FUNCTION_BLOCK FB_CassetteLoader EXTENDS FB_PackML_BaseModule

VAR
	    // Sub module definitions here

    // List of sub modules
    ipSubModules_Init : ARRAY[1..Parameters_PackML_Base.MAX_NO_OF_SUBMODULES] OF I_PackML_BaseModule := [];

    // Component definitions here
    ElevatorAxisA : FB_Component_BasicAxis := (Name := 'ElevatorA');
	ElevatorAxisB : FB_Component_BasicAxis := (Name := 'ElevatorB');
	ShuttleAxis : FB_Component_BasicAxis := (Name := 'Shuttle');
	MapSensorA : FB_DigitalSensor := (Name := 'MapSensorA');
	MapSensorB : FB_DigitalSensor := (Name := 'MapSensorB');
	
	//Assign Homing Routine to Use the Absolute Encoder, using the persistent struct below
	AbsHomingElevA : FB_HomeRoutine_AbsHoming;
	AbsHomingElevB : FB_HomeRoutine_AbsHoming;
	AbsHomingShuttle : FB_HomeRoutine_AbsHoming;
		
	//Alarms for this Module
	LoaderAlarms : ARRAY[1..LOADER_ALARM_COUNT] OF FB_TcAlarm;
	
	//Data for module
    Recipe : ST_LoaderRecipe;
	CassetteAStatus : ST_CassetteStatus;
	CassetteBStatus : ST_CassetteStatus;
	_ElevatorAxisAStagePosition : LREAL;
	_ElevatorAxisBStagePosition : LREAL;
	_ShuttleAxisStagePosition : LREAL;
	_ElevatorAxisAHomePosition : LREAL;
	_ElevatorAxisBHomePosition : LREAL;
	_ShuttleAxisHomePosition : LREAL;
	
	//HMI Control for EM
    fbControlSourceHMI : FB_ControlSource_HMI;
	
	//Load or Unload Mode: Commanded by External, TRUE= Load, FALSE = Unload
	_LoadOrUnload : BOOL;
	_ShuttleReady : BOOL;

	//This trigger each axis at the abs zero position when in maintenance or manual mode
	AbsHomeCmdA: BOOL;
	AbsHomeCmdB: BOOL;
	AbsHomeCmdShuttle: BOOL;
	_NeedsMapping: BOOL;
	_NextSlot: DINT;
	_NextCassette: INT;
END_VAR

VAR CONSTANT
	LOADER_ALARM_COUNT : INT := 6;
END_VAR

VAR PERSISTENT
	ElevAHomingParameters : ST_AbsHomeParameters;
	ElevBHomingParameters : ST_AbsHomeParameters;
	ShuttleHomingParameters : ST_AbsHomeParameters;
END_VAR

ShuttleHomingParameters.PositionBias := 0;

METHOD PROTECTED Aborting
VAR_INPUT
END_VAR
CASE SequenceState OF
    0:
        NoStateTasksToComplete := FALSE;
        SequenceState          := SequenceState + 10;
    10:
        ElevatorAxisA.Stop();
		ElevatorAxisB.Stop();
		ShuttleAxis.Stop();
//        IF (ElevatorAxisA.Stopped AND ElevatorAxisB.Stopped AND ShuttleAxis.Stopped) THEN
//            SequenceState := SequenceState + 10;
//        END_IF
		SequenceState := SequenceState + 10;
    20:
        // Disable here
        ElevatorAxisA.Disable();
		ElevatorAxisB.Disable();
		ShuttleAxis.Disable();

        // Check not enabled here
        IF NOT (ElevatorAxisA.Enabled AND ElevatorAxisB.Enabled AND ShuttleAxis.Enabled) THEN
            SequenceState := SequenceState + 10;
        END_IF
    30:
        StateTasksComplete := TRUE;
END_CASE

SUPER^.Aborting();
END_METHOD

PROPERTY BladeThickness : LREAL
GET
BladeThickness := recipe.Elevator.BladeThickness;
END_GET
SET
BladeThickness := recipe.Elevator.BladeThickness;
END_SET
END_PROPERTY

PROPERTY CassettePitch : LREAL
GET
CassettePitch := recipe.Elevator.CassettePitch;
END_GET
SET
recipe.Elevator.CassettePitch := CassettePitch;
END_SET
END_PROPERTY

PROPERTY CassetteSlotHeight : LREAL
GET
CassetteSlotHeight := recipe.Elevator.CassetteSlotHeight;
END_GET
SET
recipe.Elevator.CassetteSlotHeight := CassetteSlotHeight;
END_SET
END_PROPERTY

PROPERTY CassetteSlotNumber : INT
GET
CassetteSlotNumber := recipe.Elevator.CassetteSlotNumber;
END_GET
SET
recipe.Elevator.CassetteSlotNumber := CassetteSlotNumber;
END_SET
END_PROPERTY

METHOD PROTECTED Clearing
VAR_INPUT
END_VAR
CASE SequenceState OF
    0:
        NoStateTasksToComplete := FALSE;
        SequenceState          := SequenceState + 10;
	10:
        //Reset any alarms that get latched
        //PullWheelAlarms[E_PullWheels.StartTimeout].Clear(0, 0);
        SequenceState := SequenceState + 10;
    20:
        StateTasksComplete := TRUE;
END_CASE

SUPER^.Clearing();
END_METHOD

METHOD CyclicLogic
VAR_INPUT
END_VAR

VAR
	i : INT;
	TotalInCassetteA : INT;
	TotalInCassetteB : INT;
	CassetteAInteger : ARRAY[0..23] OF INT; //matching array with INT type
	CassetteBInteger : ARRAY[0..23] OF INT; //matching array with INT type
END_VAR
IF NOT _InitComplete THEN
    _InitComplete := Initialize();
    RETURN;
END_IF

SUPER^.CyclicLogic();

//Set the current alarm severity for this module
_CurrentAlarmSeverity   := F_GetMaxSeverityRaised(Alarms := LoaderAlarms, CurrentSeverity := _CurrentAlarmSeverity);

//Add up the number of waveguides in each cassette and mark the cassette status as full
	FOR i := 0 TO 23 DO
		IF CassetteAStatus.WaveguidePresent[i] = TRUE THEN
			CassetteAInteger[i] := 1;
		ELSE
			CassetteAInteger[i] := 0;
		END_IF
		TotalInCassetteA := TotalInCassetteA + CassetteAInteger[i];
		IF TotalInCassetteA > 22 THEN
			CassetteAStatus.CassetteFull := TRUE;
		END_IF
	END_FOR; 
	
	FOR i := 0 TO 23 DO
		IF CassetteBStatus.WaveguidePresent[i] = TRUE THEN
			CassetteBInteger[i] := 1;
		ELSE
			CassetteBInteger[i] := 0;
		END_IF
		TotalInCassetteB := TotalInCassetteB + CassetteBInteger[i];
		IF TotalInCassetteB > 22 THEN
			CassetteBStatus.CassetteFull := TRUE;
		END_IF
	END_FOR;
END_METHOD

METHOD DetermineNextSlot : DINT
VAR_INPUT
	CassetteID : ST_CassetteStatus;
END_VAR

VAR
	i: DINT;
END_VAR
//This method searches the wafer map array from the bottom to the top, returning the highest slot that is empty
	FOR i := 0 TO 23 DO
		IF CassetteID.WaveguidePresent[i] = FALSE THEN
			DetermineNextSlot := i;
		END_IF
	END_FOR;
END_METHOD

METHOD DetermineNextWaveguide : INT
VAR_INPUT
		CassetteID : ST_CassetteStatus;
END_VAR

VAR
	i: INT;
END_VAR
//This method searches the wafer map array from the bottom to the top, returning the lowest slot that is full
	FOR i := 23 TO 0 DO
		IF CassetteID.WaveguidePresent[i] = TRUE THEN
			DetermineNextWaveguide := i;
		END_IF
	END_FOR;
END_METHOD

PROPERTY ElevatorAcceleration : LREAL
GET
ElevatorAcceleration := recipe.Elevator.Acceleration;
END_GET
SET
recipe.Elevator.Acceleration := ElevatorAcceleration;
END_SET
END_PROPERTY

PROPERTY ElevatorFirstWaveguidePosition : LREAL
GET
ElevatorFirstWaveguidePosition := recipe.Elevator.FirstWaveguidePosition;
END_GET
SET
recipe.Elevator.FirstWaveguidePosition := ElevatorFirstWaveguidePosition;
END_SET
END_PROPERTY

PROPERTY ElevatorVelocity : LREAL
GET
ElevatorVelocity := recipe.Elevator.Velocity;
END_GET
SET
recipe.Elevator.Velocity := ElevatorVelocity;
END_SET
END_PROPERTY

METHOD PROTECTED Execute
VAR_INPUT
END_VAR
CASE _CurrentMode OF
    //=================================PRODUCTION MODE==================================
    E_PMLUnitMode.ePMLUnitMode_Production:
		IF _LoadOrUnload = TRUE THEN // _LoadOrUnload = TRUE means LOAD the cassette
			
		//Loading case
			CASE SequenceState OF

				10:		//Figure out where to put the next waveguide
						//we will load cassette A (top-down) before cassette B (top-down), so if A is full start loading B 
						IF NOT CassetteAStatus.CassetteFull THEN
							_NextSlot := DetermineNextSlot(CassetteID := CassetteAStatus);
							_NextCassette := 0; 
						ELSE	
							_NextSlot := DetermineNextSlot(CassetteID := CassetteBStatus);
							_NextCassette := 1;
						END_IF
						SequenceState := SequenceState + 10;
				20:		//Make sure that the space under/over the slot is clear, abort if obstructed
						IF _NextCassette = 0 THEN
							IF (CassetteAStatus.ClearBelowWaveguide[_NextSlot] AND CassetteAStatus.ClearBelowWaveguide[_NextSlot + 1]) = TRUE THEN
								SequenceState := SequenceState + 10;
							ELSE
								//changestate(ePMLState_Aborting);
							END_IF
						ELSE
							IF (CassetteBStatus.ClearBelowWaveguide[_NextSlot] AND CassetteBStatus.ClearBelowWaveguide[_NextSlot + 1]) = TRUE THEN
								SequenceState := SequenceState + 10;
							ELSE
								//changestate(ePMLState_Aborting);
							END_IF
						END_IF
						SequenceState := SequenceState + 10;
				30: 	//Move all to staged position
						SequenceState := SequenceState + 10;
				40:		//Call PlaceToNextOpenSlot method
						PlaceToNextOpenSlot(_NextCassette, _NextSlot);
						SequenceState := SequenceState + 10;
				50:		//Depending on which cassette we loaded, update the map to add the waveguide:
						IF _NextCassette = 0 THEN
							CassetteAStatus.WaveguidePresent[_NextSlot]:= 1;
						ELSE
							CassetteBStatus.WaveguidePresent[_NextSlot]:= 1;
						END_IF
						SequenceState := SequenceState + 10;

				99:		//based on the cassette status, either go into suspending or completing
						IF (CassetteAStatus.CassetteFull AND CassetteBStatus.CassetteFull) THEN
							StateComplete();
						ELSE
							//go into suspending state
							//changestate(ePMLState_Suspending);
						END_IF
			END_CASE
			
		//Unload Case	
		ELSE //_LoadOrUnload = FALSE means UNLOAD the cassette
			
			CASE SequenceState OF
				10: //Figure out which waveguide to remove first
				//we will unload cassette A (bottom-up) before cassette B (bottom-up), so if A is empty start unloading B
						IF CassetteAStatus.CassetteFull THEN
							_NextSlot := DetermineNextWaveguide(CassetteID := CassetteAStatus);
							_NextCassette := 0; 
						ELSE	
							_NextSlot := DetermineNextWaveguide(CassetteID := CassetteBStatus);
							_NextCassette := 1;
						END_IF
						SequenceState := SequenceState + 10;
				20:		//Make sure that the space under/over the slot is clear, abort if obstructed
						IF _NextCassette = 0 THEN
							IF (CassetteAStatus.ClearBelowWaveguide[_NextSlot] AND CassetteAStatus.ClearBelowWaveguide[_NextSlot + 1]) = TRUE THEN
								SequenceState := SequenceState + 10;
							ELSE
								//changestate(ePMLState_Aborting);
							END_IF
						ELSE
							IF (CassetteBStatus.ClearBelowWaveguide[_NextSlot] AND CassetteBStatus.ClearBelowWaveguide[_NextSlot + 1]) = TRUE THEN
								SequenceState := SequenceState + 10;
							ELSE
								//changestate(ePMLState_Aborting);
							END_IF
						END_IF
						SequenceState := SequenceState + 10;
				30:		//Pre-position the stages
						IF _NextCassette = 0 THEN
							ElevatorAxisA.MoveAbsolute(_ElevatorAxisAStagePosition,TRUE);
							ElevatorAxisB.MoveAbsolute(_ElevatorAxisBHomePosition,TRUE);
							ShuttleAxis.MoveAbsolute(_ShuttleAxisStagePosition, TRUE);
						ELSE
							ElevatorAxisA.MoveAbsolute(_ElevatorAxisAHomePosition,TRUE);
							ElevatorAxisB.MoveAbsolute(_ElevatorAxisBStagePosition,TRUE);
							ShuttleAxis.MoveAbsolute(_ShuttleAxisStagePosition, TRUE);
						END_IF
						SequenceState := SequenceState + 10;
				40: 	//Confirm all axis preposition movements are complete
						IF (ElevatorAxisA.Busy AND ElevatorAxisB.Busy AND ShuttleAxis.Busy) THEN
							SequenceState := SequenceState + 10;
						END_IF
				50:		//Call GetNextWaveguide method
						GetNextWaveGuide(_NextCassette, _NextSlot);
						SequenceState := SequenceState + 10;
				60:		//Depending on which cassette we unloaded, update the map to remove the waveguide:
						IF _NextCassette = 0 THEN
							CassetteAStatus.WaveguidePresent[_NextSlot]:= 0;
						ELSE
							CassetteBStatus.WaveguidePresent[_NextSlot]:= 0;
						END_IF
						SequenceState := SequenceState + 10;
				
			END_CASE
		END_IF
//If we are waiting for the tool to load/unload the waveguide, switch to Suspending state



    //=================================MAINTENANCE & MANUAL MODE==================================		
    E_PMLUnitMode.ePMLUnitMode_Maintenance, E_PMLUnitMode.ePMLUnitMode_Manual:
        //Reset the abs zero position when commanded
		IF AbsHomeCmdA THEN
    		AbsHomingElevA.Execute();
    		AbsHomeCmdA:=FALSE;
		END_IF;
		
		IF AbsHomeCmdB THEN
    		AbsHomingElevA.Execute();
    		AbsHomeCmdB:=FALSE;
		END_IF;
		
		IF AbsHomeCmdShuttle THEN
    		AbsHomingElevA.Execute();
    		AbsHomeCmdShuttle:=FALSE;
		END_IF;
END_CASE
END_METHOD

METHOD GetNextWaveguide : BOOL
VAR_INPUT
	NextCassette : INT;
	NextSlot : DINT;
END_VAR
//This method will get the waveguide in the cassette and slot defined as next-available and move the shuttle to the tool position
END_METHOD

//! @summary Basic module initialization logic
METHOD PROTECTED Initialize : BOOL;
VAR
	i						 : UDINT;
	varInfo					 : __SYSTEM.VAR_INFO;
	AllSubUnitsInitialized	 : BOOL := TRUE;
	AllComponentsInitialized : BOOL := TRUE;
END_VAR

//! @description This method is called by <c>CyclicLogic()</c> as required
Initialize := FALSE;
CASE DescendantSequenceState OF
    0:
		//RegisterComponent here (none for now)
        _LogModeChanges         := FALSE;
        _LogStateChanges        := FALSE;
        DescendantSequenceState := DescendantSequenceState + 10;
    10:
        //Setup Custom modes here
        CustomModes(eMode                          :=,
                    sName                          := 'Name',
                    bDisableClearing               := FALSE,
                    bDisableStarting               := FALSE,
                    bDisableSuspended              := FALSE,
                    bDisableStopping               := FALSE,
                    bDisableAborting               := FALSE,
                    bDisableHolding                := TRUE, //no operator hold state 
                    bDisableHeld                   := TRUE,
                    bDisableUnholding              := TRUE,
                    bDisableSuspending             := FALSE,
                    bDisableUnsuspending           := FALSE,
                    bDisableResetting              := FALSE,
                    bDisableIdle                   := FALSE,
                    bDisableCompleting             := FALSE,
                    bDisableComplete               := FALSE,
                    bEnableUnitModeChangeStopped   := TRUE,
                    bEnableUnitModeChangeIdle      := TRUE,
                    bEnableUnitModeChangeSuspended := FALSE,
                    bEnableUnitModeChangeExecute   := FALSE,
                    bEnableUnitModeChangeAborted   := FALSE,
                    bEnableUnitModeChangeHeld      := FALSE,
                    bEnableUnitModeChangeComplete  := FALSE,
                    bError                         =>,
                    nErrorId                       =>);
        DescendantSequenceState := DescendantSequenceState + 10;
    20:
        //Copy Mode names
        FOR i := 1 TO 3 DO
            ModeNames[i] := F_UnitModeToString(UDINT_TO_DINT(i));
        END_FOR

        //Initialize_TagData();
		RegisterExternalController(Controller := fbControlSourceHMI);
		fbControlSourceHMI.CyclicLogic();
        DescendantSequenceState := DescendantSequenceState + 10;
		
	30: //Register homing methods for each axis
//				ShuttleAxis.HomeMethod := AbsHomingShuttle;
//				AbsHomingShuttle.Parameters := ShuttleHomingParameters;
//				ElevatorAxisA.HomeMethod := AbsHomingElevA;
//				AbsHomingElevA.Parameters := ElevAHomingParameters;
//				ElevatorAxisB.HomeMethod := AbsHomingElevB;
//				AbsHomingElevB.Parameters := ElevBHomingParameters;
      	DescendantSequenceState := DescendantSequenceState + 10;
    40:
        //Call the Super
        IF SUPER^.Initialize() THEN
            DescendantSequenceState := DescendantSequenceState + 10;
        END_IF
    50:
        Initialize := TRUE;
END_CASE
END_METHOD

METHOD LoadCassette : BOOL
VAR_INPUT

END_VAR
(* This method will allow the user to stop the machine, open the door, install cassettes, 
close the door, restart the machine, map the cassettes and go into a ready state *)
END_METHOD

PROPERTY LoadOrUnload : bool
GET
LoadOrUnload := _LoadOrUnload;
END_GET
SET
_LoadOrUnload := LoadOrUnload;
END_SET
END_PROPERTY

METHOD MapCassette : BOOL
VAR_INPUT
	CassetteToMap : INT; //Cassette A is zero, Cassette B is one, etc.
END_VAR

VAR
	
END_VAR

//this method will map the cassette specified in CassetteToMap, saving the output in the array CassetteAStatus.WaveguidePresent
END_METHOD

METHOD PlaceToNextOpenSlot : BOOL
VAR_INPUT
	NextCassette : INT;
	NextSlot : DINT;
END_VAR
//This method will place the waveguide (placed on the blade by the tool) to the next open slot
END_METHOD

METHOD PROTECTED Resetting
VAR_INPUT
END_VAR
CASE _CurrentMode OF
    //=================================PRODUCTION MODE==================================
    E_PMLUnitMode.ePMLUnitMode_Production:
        CASE SequenceState OF
            0:
                NoStateTasksToComplete := FALSE;
                SequenceState          := SequenceState + 10;
            10:
				// Enable here
				ElevatorAxisA.Enable();
				ElevatorAxisB.Enable();
				ShuttleAxis.Enable();	
				// Check enabled here
				IF (ElevatorAxisA.Enabled AND ElevatorAxisB.Enabled AND ShuttleAxis.Enabled) THEN
					StateTasksComplete := TRUE;
				END_IF
                //SequenceState := SequenceState + 10;
            20:
                //IF (*LeftPullWheel.InGear AND*) RightPullWheel.InGear THEN
                    //StateTasksComplete := TRUE;
                //END_IF
        END_CASE

    //=================================MAINTENANCE & MANUAL MODE==================================	
    E_PMLUnitMode.ePMLUnitMode_Maintenance, E_PMLUnitMode.ePMLUnitMode_Manual:
        ;
END_CASE

SUPER^.Resetting();
END_METHOD

PROPERTY ShuttleCassettePosition : LREAL
GET
ShuttleCassettePosition := recipe.Shuttle.CassettePosition;
END_GET
SET
recipe.Shuttle.CassettePosition := ShuttleCassettePosition;
END_SET
END_PROPERTY

PROPERTY ShuttleReady : BOOL
GET
ShuttleReady := _ShuttleReady;
END_GET
SET
_ShuttleReady := ShuttleReady;
END_SET
END_PROPERTY

PROPERTY ShuttleToolPosition : LREAL
GET
ShuttleToolPosition := recipe.Shuttle.ToolPosition;
END_GET
SET
recipe.Shuttle.ToolPosition := ShuttleToolPosition;
END_SET
END_PROPERTY

PROPERTY ShuttleVelocity : LREAL
GET
ShuttleVelocity := recipe.Shuttle.Velocity;
END_GET
SET
recipe.Shuttle.Velocity := ShuttleVelocity;
END_SET
END_PROPERTY

//! @summary This method contains code which will execute when this PackML module is in the <b>Starting</b> state
METHOD PROTECTED Starting
VAR
	i				: UDINT;
	SubModulesReady : BOOL := TRUE;
END_VAR

(*! <description><b></b><table> 
	<tr>
		<th> Previous State </th>
		<th> Transition In </th>
		<th> Transition Out </th>
		<th> Next State  </th> 
	</tr>
	<tr>
		<td> Idle </td>
		<td> Start Command </td> 
		<td> State Complete </td>
		<td> Execute </td> 
	</tr>
</table>
This method is called as required by <c>StateControl()</c>
</description> 

*)
CASE _CurrentMode OF
    //=================================PRODUCTION MODE==================================
    E_PMLUnitMode.ePMLUnitMode_Production:
        CASE SequenceState OF
            0:
                NoStateTasksToComplete := FALSE;
                SequenceState          := SequenceState + 10;
            10:
                //assign all recipe values here
				ElevatorAxisA.Velocity := Recipe.Elevator.Velocity;
				ElevatorAxisA.Acceleration := Recipe.Elevator.Acceleration;
                SequenceState := SequenceState + 10;
			20:
				//Home the shuttle axis
				ShuttleAxis.Home();
				SequenceState := SequenceState + 10;
			30: 
				//Home the elevator axis at the same time
				ElevatorAxisA.Home();
				ElevatorAxisB.Home();
				SequenceState := SequenceState + 10;
			40: //With the elevator stages at home, map each cassette
				MapCassette(0);
				IF NOT ElevatorAxisA.Busy THEN
					SequenceState := SequenceState + 10;
				END_IF
			50: //
				MapCassette(1);
				IF NOT ElevatorAxisB.Busy THEN
					SequenceState := SequenceState + 10;
				END_IF
            60:
				//Verify that home is completed and home sensors are satisfied
                IF NOT (ElevatorAxisA.Busy AND ElevatorAxisB.Busy AND ShuttleAxis.Busy) THEN
                    StateTasksComplete := TRUE;
                END_IF
        END_CASE

    //=================================MAINTENANCE & MANUAL MODE==================================
    E_PMLUnitMode.ePMLUnitMode_Maintenance, E_PMLUnitMode.ePMLUnitMode_Manual:
        ;
END_CASE
END_METHOD

METHOD PROTECTED Stopping
VAR_INPUT
END_VAR
CASE _CurrentMode OF
    //=================================PRODUCTION MODE==================================
	//	The elevators and shuttle are disabled, so they can not be moved. Does this state do anything?
	
    E_PMLUnitMode.ePMLUnitMode_Production:
        CASE SequenceState OF
            0:
                NoStateTasksToComplete := FALSE;
                //PullWheelCylinder.Retract();
                SequenceState := SequenceState + 10;
            10:
				
//                IF PullWheelCylinder.Retracted THEN
//                    SequenceState := SequenceState + 10;
//                END_IF
				SequenceState := SequenceState + 10;
            20:
                StateTasksComplete := TRUE;
        END_CASE

    //=================================MAINTENANCE & MANUAL MODE==================================
    E_PMLUnitMode.ePMLUnitMode_Maintenance, E_PMLUnitMode.ePMLUnitMode_Manual:
        ;
END_CASE

SUPER^.Stopping();
END_METHOD

//! @summary This method contains code which will execute when this PackML module is in the <b>Suspending</b> state
METHOD PROTECTED Suspending
VAR
	i				: UDINT;
	SubModulesReady : BOOL := TRUE;
END_VAR

(*! <description><b>Note:</b> The <i>Suspend</i> command is intended to be initiated by automatic detection of upstream/downstream jams, etc. It is meant to be distinct from a <i>Hold</i> in that <i>Hold</i> should be commanded by an operator.  Both <i>Hold</i>and<i>Suspend</i> result in a <i>paused</i> state which should allow resumption of the <b>Execute</b> state. 
<table> 
	<tr>
		<th> Previous State </th>
		<th> Transition In </th>
		<th> Transition Out </th>
		<th> Next State  </th> 
	</tr>
	<tr>
		<td> Execute </td>
		<td> Suspend Command </td> 
		<td> State Complete </td>
		<td> Suspended </td> 
	</tr>
</table>
This method is called as required by <c>StateControl()</c>
</description> 

*)
//Notify the tool that the shuttle is waiting
END_METHOD

METHOD UnloadCassette : BOOL
VAR_INPUT
END_VAR
(* This method will allow the user to trigger an unload sequence, open the door, remove the cassettes,
close the door and wait for new cassettes *)
END_METHOD

PROPERTY WaveguideThickness : LREAL
GET
WaveguideThickness := recipe.Elevator.WaveguideThickness;
END_GET
SET
recipe.Elevator.WaveguideThickness := WaveguideThickness;
END_SET
END_PROPERTY

END_FUNCTION_BLOCK

(* stored: Version 1.1.0.1, ProductVersion 3.1.4024.12
   POU FB_CassetteLoader: Id {e1442105-7e9e-435d-a38b-588b19f392f0}, SpecialFunc None
   Folder I_CyclicFB: Id {ab7f0c2a-9be7-47f0-880e-086853a8a382}
   Folder Methods: Id {7d33ab3d-f7f6-49cb-81a8-db41b285a909}
   Folder Acting States: Id {4dc4a433-6b0f-4a50-87a1-2e14bd3ee869}
   Folder Custom Methods: Id {c87beed5-5d3b-4fd7-b255-b9a95be15bb8}
   Folder Waiting States: Id {4ade595e-9a9e-4bb8-8687-f1fd8755933b}
   Folder Properties: Id {0f5023fd-9dc3-438b-8401-c69763c4d630}
   Method Aborting: Id {33e9e90e-3c8f-4146-b67b-b2569e47f20a}
   Property BladeThickness: Id {9b89bbfa-aeab-4504-a73f-51ef9aacf01e}
   Get Get: Id {7e38671f-1374-4a26-a08f-91a1b03491a2}
   Set Set: Id {8de687c7-47ef-4748-96b6-a06c87012404}
   Property CassettePitch: Id {99b231eb-d7c5-4fb1-9e23-58eaa7f6727c}
   Get Get: Id {e55fadb5-c9db-4ee9-8fa1-306a0bafd3f8}
   Set Set: Id {866448cc-784e-4b68-8e27-c18b16ca3ceb}
   Property CassetteSlotHeight: Id {066cae7e-2874-46c9-a619-7f2e4bdb666c}
   Get Get: Id {7f9e9967-649e-4a92-b0ae-f6dd4378639c}
   Set Set: Id {1c704c35-c70b-493b-81a6-11eb3fac4214}
   Property CassetteSlotNumber: Id {7e3fa52a-5f57-4861-aec1-955bb5ec4fa4}
   Get Get: Id {4bb2f4dd-5aff-4203-a947-393b27ff1f15}
   Set Set: Id {0bb09dad-87b2-456d-8868-340314efe1e4}
   Method Clearing: Id {d98b2f50-4364-48fd-8d94-31f4c0da6c04}
   Method CyclicLogic: Id {b8b1f610-e7ce-489d-abc2-e340ab00a953}
   Method DetermineNextSlot: Id {1346f1ec-1877-4d3d-ad4d-af6d28eb70b2}
   Method DetermineNextWaveguide: Id {6de7ea29-ee39-4576-ae0e-b4af486f76c4}
   Property ElevatorAcceleration: Id {ec23dba9-1f3d-44ba-8976-3d1b29c1b0e7}
   Get Get: Id {6585a2df-20c2-4b7b-90cd-d477bf988a55}
   Set Set: Id {3a1f2b02-b519-4bae-9de0-393d4f0d03d8}
   Property ElevatorFirstWaveguidePosition: Id {d49b5647-3a4e-4c76-9ca2-fc0bd2b4cc85}
   Get Get: Id {06ed25cb-d6c8-48d1-aa1f-9d96edd75fc9}
   Set Set: Id {a5056d01-f334-418b-984c-c642c9304f6d}
   Property ElevatorVelocity: Id {596ec064-d93a-4634-b242-badec1e1af24}
   Get Get: Id {1d423af7-4da4-4783-982a-cb398b3f1bab}
   Set Set: Id {a5358478-4863-490b-964e-0a374995c995}
   Method Execute: Id {f9997ab5-bbbe-4198-ab99-4b129008096f}
   Method GetNextWaveguide: Id {1997f330-ca7f-4a4e-8e23-7984b89fe323}
   Method Initialize: Id {dc16f921-5111-486b-8d1c-42cc395f7e89}
   Method LoadCassette: Id {ee35de60-c5f2-4af1-8448-c7a13c5e4bd2}
   Property LoadOrUnload: Id {e8d97373-1153-461a-aa4f-8058a8edfe0d}
   Get Get: Id {fb526f32-c36d-4263-9bbf-27c96a94bcee}
   Set Set: Id {29b02b2c-0edd-4400-9325-52589c8ca530}
   Method MapCassette: Id {56a6e915-6f8a-4fb4-ad24-df0b01475ae7}
   Method PlaceToNextOpenSlot: Id {df984bf4-69c9-4aed-ad44-c7461d2d7919}
   Method Resetting: Id {111af2e3-4fe9-4e0f-9563-9b8550596a16}
   Property ShuttleCassettePosition: Id {86ad11d0-eab7-4f1a-9cfc-1c216e256605}
   Get Get: Id {07de01f3-c991-4ce6-aea1-124bf272898f}
   Set Set: Id {16f2069d-2392-4aac-9ff6-a6575f31f614}
   Property ShuttleReady: Id {9d53f2e7-2f58-409e-87c1-9367c222f1d7}
   Get Get: Id {c8d78756-68d5-43c5-a438-cb87dd60f352}
   Set Set: Id {b8c85d81-3b12-44d9-aba4-78ec55859cf3}
   Property ShuttleToolPosition: Id {d9c4f83d-a087-4177-8e75-79e642b536e5}
   Get Get: Id {6231cdc5-356f-4940-89b0-7e214191d0b3}
   Set Set: Id {fd9bed83-13be-4030-b114-1537baf9f9f9}
   Property ShuttleVelocity: Id {35d9c7f6-51f0-4e07-8604-e69c2eca9451}
   Get Get: Id {48d75316-5457-4a47-bbfb-4bfd39d36374}
   Set Set: Id {70b67659-7aab-445b-a7d1-b79d1d645663}
   Method Starting: Id {58998f7f-7f9d-4d33-84bd-cff353cfff86}
   Method Stopping: Id {0e458215-351e-44f5-9214-989717195c78}
   Method Suspending: Id {77b8e905-0e66-474d-952e-699895a2e113}
   Method UnloadCassette: Id {8aea1982-41d3-46b5-96ee-f96fdba3f914}
   Property WaveguideThickness: Id {229efe54-3fa5-464a-aa50-fa72bcb3a290}
   Get Get: Id {b679666f-fa70-4b69-a334-687177986088}
   Set Set: Id {3fd9057d-0e65-431d-8eb7-1800583dfa1b} *)
